FUNCTION_BLOCK FB_Alarm IMPLEMENTS I_Logger
VAR_INPUT
END_VAR
VAR_OUTPUT
END_VAR
VAR
	nLength:		INT;
	aEvent:			ARRAY [0..nMax] OF ST_Event;
END_VAR
VAR CONSTANT
	nMax:			INT:= 99;
END_VAR

METHOD M_Find : DINT
VAR_INPUT
	stEvent	: 		ST_Event;
END_VAR
VAR
	nIndex: 	DINT;
END_VAR
// Object already in List
M_Find := -1;
WHILE nIndex < nLength DO
    IF (aEvent[nIndex].Source = stEvent.Source) 
		AND_THEN (aEvent[nIndex].EventType = stEvent.EventType) 
		AND_THEN (aEvent[nIndex].Message = stEvent.Message) THEN
			M_Find := nIndex;
			RETURN;
    END_IF
	nIndex := nIndex + 1;
END_WHILE
END_METHOD

METHOD M_Log
VAR_INPUT
	stEvent	: 		ST_Event;
END_VAR

VAR
	nIndex: DINT;
END_VAR
IF (nIndex:= M_Find(stEvent)) = -1 THEN
	aEvent[nLength]:= stEvent;
	nLength:= nLength + 1;
ELSE
	aEvent[nIndex]:= stEvent;	
END_IF
END_METHOD

END_FUNCTION_BLOCK

(* stored: Version 1.1.0.1, ProductVersion 3.1.4024.12
   POU FB_Alarm: Id {6b962909-8df1-4dcd-be8b-465f6b091a91}, SpecialFunc None
   Method M_Find: Id {1cfa321c-140c-45bd-9dda-bac3538adfc3}
   Method M_Log: Id {22357804-3270-478e-9b42-7d8931f13ab7} *)
